Fanuc KAREL source: FRAME.kl

PROGRAM T
%NOLOCKGROUP
VAR
 v0 : POSITION
 v1 : POSITION
 v2 : POSITION
 v3 : POSITION
 res : POSITION
BEGIN
 res = FRAME(v0, v1, v2, v3)
END T
